(* PLC project Untitled1, Beckhoff Automation GmbH TF6420 Database Server Query Analyser 1.0.0.0 *)
(* stored: creationDateTime 2020-05-17T15:27:27, modificationDateTime 2020-05-17T15:27:27 *)

TYPE test : STRUCT
  ID : DINT;
  Feld1 : DINT;
END_STRUCT;
END_TYPE
